TYPE ExampleDomain_Io_Out :
STRUCT
END_STRUCT
END_TYPE

(* stored: Version 1.1.0.1
   DUT ExampleDomain_Io_Out: Id {f56c954d-73c2-431c-b49d-98f0848af0a7} *)
